Yaskawa INFORM job: X2_55B(90,0).JBI

/JOB
//NAME X2_55B(90,0)
//POS
///NPOS 394,394,394,16,0,0
///TOOL 0
///POSTYPE PULSE
///PULSE
C00000=3322,-122452,-100913,-73,83322,449
C00001=-186633,-49441,-49230,37711,87728,-55120
C00002=-175086,-27134,-34976,36439,84930,-51244
C00003=-172101,-26870,-32446,36082,82517,-50807
C00004=-170908,-26670,-31367,35943,81558,-50627
C00005=-169791,-28532,-32653,35785,80956,-50361
C00006=-170908,-26670,-31367,35943,81558,-50627
C00007=-170104,-28160,-32639,35819,81236,-50399
C00008=-170107,-27903,-30796,35900,80418,-50669
C00009=-170104,-28160,-32639,35819,81236,-50399
C00010=-170752,-27064,-31161,35943,81224,-50672
C00011=-169656,-24122,-29101,35757,80964,-50300
C00012=-170752,-27064,-31161,35943,81224,-50672
C00013=-171397,-28056,-32227,36028,81614,-50812
C00014=-174408,-28429,-34833,36375,84032,-51262
C00015=-173676,-39982,-43344,21171,57836,-56527
C00016=-171324,-36683,-38335,20265,55943,-55912
C00017=-170409,-35305,-36277,19908,55192,-55668
C00018=-170412,-34971,-34390,20145,54260,-55855
C00019=-170409,-35305,-36277,19908,55192,-55668
C00020=-170406,-35026,-34613,20115,54362,-55832
C00021=-168977,-33998,-33935,19313,54123,-55256
C00022=-170406,-35026,-34613,20115,54362,-55832
C00023=-171322,-36428,-36691,20470,55114,-56078
C00024=-173675,-39790,-41746,21371,57009,-56697
C00025=-185662,-62363,-56229,27773,58122,-61625
C00026=-182957,-37243,-22211,38142,77839,-57028
C00027=-174986,-21904,-11817,37450,75534,-54407
C00028=-172006,-20811,-8603,37402,73103,-53977
C00029=-171589,-19133,-6407,37448,72531,-54000
C00030=-170468,-20788,-7609,37359,71957,-53715
C00031=-171113,-19844,-6927,37410,72288,-53878
C00032=-171113,-19561,-6133,37473,72012,-53977
C00033=-171113,-19098,-4854,37577,71571,-54137
C00034=-171113,-19354,-5558,37520,71812,-54050
C00035=-170785,-16593,-3525,37458,71805,-53909
C00036=-169831,-14075,-1633,37337,71498,-53600
C00037=-170747,-16496,-3451,37453,71794,-53895
C00038=-172938,-18790,-5592,37628,72854,-54473
C00039=-174418,-22969,-11095,37549,74492,-54531
C00040=-173590,-36455,-27464,23265,50415,-58157
C00041=-171241,-32608,-21983,22436,48472,-57522
C00042=-170327,-31009,-19725,22109,47697,-57271
C00043=-170330,-30281,-17521,22452,46786,-57499
C00044=-170327,-31009,-19725,22109,47697,-57271
C00045=-170446,-30448,-17835,22480,46917,-57523
C00046=-169016,-29467,-17169,21618,46622,-56894
C00047=-170446,-30448,-17835,22480,46917,-57523
C00048=-171361,-32070,-20116,22801,47697,-57774
C00049=-173714,-35969,-25651,23617,49653,-58408
C00050=-187157,-59404,-40892,31105,51702,-64292
C00051=-182523,-36435,-21722,38111,77739,-56877
C00052=-175053,-21948,-11876,37454,75574,-54422
C00053=-172072,-20861,-8666,37406,73142,-53992
C00054=-170880,-20336,-7310,37391,72173,-53819
C00055=-169763,-22108,-8585,37302,71589,-53539
C00056=-170880,-20336,-7310,37391,72173,-53819
C00057=-163968,-30963,-18249,28546,65432,-52550
C00058=-163972,-30194,-16010,28759,64566,-52785
C00059=-171828,-19900,-6902,37491,72561,-54096
C00060=-170589,-16767,-4601,37336,72180,-53691
C00061=-169762,-14573,-2957,37230,71916,-53424
C00062=-170465,-16446,-4362,37321,72141,-53651
C00063=-172082,-18613,-7207,37365,73353,-53922
C00064=-174410,-22968,-11093,37549,74488,-54529
C00065=-173630,-36453,-27441,23290,50415,-58176
C00066=-171279,-32607,-21961,22462,48470,-57541
C00067=-170365,-31009,-19703,22136,47695,-57290
C00068=-170369,-30280,-17499,22478,46784,-57519
C00069=-170365,-31009,-19703,22136,47695,-57290
C00070=-170401,-30398,-17823,22448,46922,-57500
C00071=-168973,-29415,-17155,21586,46628,-56872
C00072=-170401,-30398,-17823,22448,46922,-57500
C00073=-171316,-32020,-20104,22769,47702,-57751
C00074=-173667,-35921,-25640,23585,49656,-58385
C00075=-184061,-55077,-38542,29439,51265,-62922
C00076=-181525,-34817,-20609,38049,77416,-56562
C00077=-175168,-22294,-12057,37473,75570,-54473
C00078=-172179,-21211,-8851,37428,73136,-54041
C00079=-164934,-20244,-11943,27524,72736,-50675
C00080=-164934,-19832,-10624,27608,72202,-50807
C00081=-164934,-20244,-11943,27524,72736,-50675
C00082=-170788,-19176,-6081,37413,72004,-53840
C00083=-170137,-20123,-6769,37360,71672,-53674
C00084=-170788,-19176,-6081,37413,72004,-53840
C00085=-170451,-17518,-5131,37330,72072,-53666
C00086=-169581,-15212,-3412,37215,71799,-53383
C00087=-170948,-17530,-5209,37372,72321,-53796
C00088=-174379,-22994,-11157,37542,74495,-54513
C00089=-173696,-36532,-27476,23332,50416,-58207
C00090=-171343,-32688,-21999,22504,48471,-57571
C00091=-170428,-31090,-19742,22178,47695,-57320
C00092=-170432,-30361,-17538,22521,46785,-57549
C00093=-170428,-31090,-19742,22178,47695,-57320
C00094=-170423,-30483,-17896,22460,46929,-57509
C00095=-168993,-29501,-17229,21598,46634,-56880
C00096=-170423,-30483,-17896,22460,46929,-57509
C00097=-171339,-32105,-20177,22781,47708,-57760
C00098=-173691,-36004,-25710,23598,49663,-58395
C00099=-183961,-54871,-38414,29383,51253,-62877
C00100=-182126,-35603,-21062,38091,77581,-56762
C00101=-175140,-21971,-11768,37472,75549,-54468
C00102=-172157,-20885,-8559,37428,73117,-54039
C00103=-170965,-20360,-7203,37414,72147,-53865
C00104=-169849,-22134,-8479,37326,71562,-53586
C00105=-170965,-20360,-7203,37414,72147,-53865
C00106=-165310,-29694,-17403,28817,66009,-52954
C00107=-165310,-29050,-15538,28988,65287,-53150
C00108=-171258,-19918,-6523,37477,72118,-54004
C00109=-170426,-17807,-4979,37371,71866,-53731
C00110=-169380,-15031,-2910,37233,71539,-53391
C00111=-169955,-16574,-4065,37309,71721,-53578
C00112=-171522,-16229,-3810,37460,72416,-54014
C00113=-174416,-22925,-11129,37542,74526,-54518
C00114=-173673,-36450,-27429,23316,50421,-58195
C00115=-171322,-32606,-21950,22488,48476,-57560
C00116=-170407,-31008,-19692,22162,47701,-57309
C00117=-170411,-30279,-17488,22505,46790,-57538
C00118=-170407,-31008,-19692,22162,47701,-57309
C00119=-170394,-30411,-17842,22442,46925,-57496
C00120=-168966,-29428,-17174,21580,46631,-56867
C00121=-170394,-30411,-17842,22442,46925,-57496
C00122=-171309,-32033,-20124,22763,47705,-57746
C00123=-173661,-35933,-25659,23580,49659,-58381
C00124=-177896,-47999,-50685,14899,88109,-20692
C00125=-171474,-13387,-32995,26955,87451,38414
C00126=-170968,-26590,-20653,68029,76629,42851
C00127=-168455,-24364,-16087,68284,74284,42470
C00128=-167462,-23391,-14189,68413,73355,42312
C00129=-167464,-22868,-12535,68611,73063,41980
C00130=-167462,-23391,-14189,68413,73355,42312
C00131=-167480,-22950,-12770,68584,73114,42023
C00132=-166431,-22389,-12367,68541,72426,42185
C00133=-167480,-22950,-12770,68584,73114,42023
C00134=-168474,-23944,-14688,68443,74043,42183
C00135=-170987,-26223,-19303,68160,76387,42569
C00136=-178015,-29196,-22452,68319,81266,41791
C00137=-175959,-27390,-21216,68244,79952,42141
C00138=-170916,-26575,-20647,68026,76596,42860
C00139=-168404,-24346,-16079,68281,74252,42479
C00140=-167411,-23372,-14181,68410,73322,42321
C00141=-167413,-22850,-12527,68608,73031,41989
C00142=-167411,-23372,-14181,68410,73322,42321
C00143=-167520,-22976,-12785,68586,73139,42016
C00144=-166471,-22416,-12382,68543,72450,42177
C00145=-167520,-22976,-12785,68586,73139,42016
C00146=-168514,-23970,-14702,68445,74068,42175
C00147=-171028,-26246,-19314,68163,76412,42561
C00148=-175959,-27390,-21216,68244,79952,42141
C00149=-177250,-26440,-20564,68269,80853,42004
C00150=-170954,-26577,-20655,68027,76623,42856
C00151=-168442,-24351,-16088,68281,74278,42475
C00152=-167449,-23792,-15537,68251,73591,42590
C00153=-167449,-23537,-14700,68349,73439,42422
C00154=-167449,-23792,-15537,68251,73591,42590
C00155=-166070,-22339,-14503,68155,72712,42832
C00156=-167449,-23792,-15537,68251,73591,42590
C00157=-168444,-23916,-14658,68443,74021,42185
C00158=-170956,-26197,-19274,68160,76364,42572
C00159=-177250,-26440,-20564,68269,80853,42004
C00160=-175728,-25304,-19738,68213,79861,42242
C00161=-170992,-26689,-20702,68035,76638,42839
C00162=-168478,-24463,-16136,68290,74291,42458
C00163=-167484,-23490,-14239,68419,73362,42300
C00164=-167486,-22966,-12584,68617,73070,41968
C00165=-167484,-23490,-14239,68419,73362,42300
C00166=-167481,-23030,-12848,68582,73118,42026
C00167=-166432,-22469,-12445,68539,72429,42188
C00168=-167481,-23030,-12848,68582,73118,42026
C00169=-168476,-24024,-14766,68441,74047,42186
C00170=-170989,-26302,-19378,68159,76391,42571
C00171=-175728,-25304,-19738,68213,79861,42242
C00172=-176618,-29227,-22045,73488,80077,41536
C00173=-172161,-28800,-21751,73383,76996,42032
C00174=-169385,-26618,-17509,73648,74607,41659
C00175=-167563,-23815,-14727,73682,73258,41735
C00176=-167563,-23156,-12665,73937,72973,41305
C00177=-167563,-23556,-13902,73784,73143,41560
C00178=-166501,-22641,-13252,73745,72429,41707
C00179=-167563,-23556,-13902,73784,73143,41560
C00180=-169398,-26250,-16243,73794,74434,41390
C00181=-172174,-28475,-20524,73502,76822,41766
C00182=-176618,-29227,-22045,73488,80077,41536
C00183=-177511,-5639,371,68424,86651,39750
C00184=-171440,-3456,2150,68562,82586,40567
C00185=-170157,619,6666,68653,81457,40444
C00186=-168331,1234,8338,68777,79954,40379
C00187=-168046,-2076,5678,68790,79736,40390
C00188=-167728,-5916,2555,68804,79503,40409
C00189=-167295,-9898,-598,68829,79172,40420
C00190=-166925,-12748,-2804,68854,78881,40421
C00191=-166573,-15365,-4788,68879,78593,40412
C00192=-169406,-16219,-7074,68798,80759,41235
C00193=-170164,-17729,-8787,68449,80176,51061
C00194=-175136,-9519,-2527,68339,83654,50553
C00195=-174791,2460,6527,68482,84972,40271
C00196=-171445,-3730,1370,68530,82722,40712
C00197=-169192,-1950,5863,68774,80488,40214
C00198=-167748,2520,10895,68924,79213,40058
C00199=-167367,-1794,7418,68947,78922,40075
C00200=-166938,-6982,3161,68992,77768,40277
C00201=-166250,-13921,-2117,69275,75344,44273
C00202=-165956,-15478,-3367,69159,75947,48234
C00203=-167609,-17034,-5893,68702,77907,50786
C00204=-170169,-18009,-9551,68404,80308,51201
C00205=-175223,-9646,-3183,68312,83847,50686
C00206=-174908,3052,7586,68499,84915,40106
C00207=-171434,-3401,2195,68562,82582,40568
C00208=-169182,-1586,6724,68821,80349,40067
C00209=-168625,2129,10992,68937,79702,39832
C00210=-168158,-2892,6969,68968,79346,39846
C00211=-167877,-6432,4056,69014,78297,40037
C00212=-167656,-9030,2010,69063,77269,40197
C00213=-167278,-12997,-1111,69137,75067,40567
C00214=-166927,-16034,-3407,69190,73221,40852
C00215=-166736,-17163,-4204,69214,73333,40784
C00216=-166964,-12102,-1327,68082,78867,40243
C00217=-166860,-10009,379,67974,81306,39758
C00218=-167599,-16670,-5060,68761,77774,50646
C00219=-170158,-17675,-8747,68448,80173,51063
C00220=-175928,-7987,-1318,68319,84203,50466
C00221=-174129,1419,6201,68516,84397,40216
C00222=-171443,-3483,2127,68562,82588,40566
C00223=-169190,-1670,6655,68820,80354,40066
C00224=-168618,1929,10819,68939,79695,39833
C00225=-168181,-3083,6692,68956,79389,39875
C00226=-167825,-6908,3653,69018,78263,40044
C00227=-167628,-9346,1685,69056,77267,40218
C00228=-167197,-13163,-1220,69143,75004,40568
C00229=-166871,-15927,-3321,69191,73184,40859
C00230=-166710,-17179,-4282,69204,73330,40804
C00231=-166618,-17311,-4405,69161,75321,40414
C00232=-167253,-2768,6900,68495,85595,38662
C00233=-167607,-16752,-5121,68762,77778,50643
C00234=-170167,-17757,-8807,68449,80178,51060
C00235=-175992,-7969,-1304,68317,84246,50458
C00236=-174493,2196,6858,68508,84639,40165
C00237=-171437,-3428,2172,68562,82584,40568
C00238=-169184,-1614,6701,68820,80351,40067
C00239=-168608,2565,11412,68945,79676,39815
C00240=-168131,-2876,6882,68959,79351,39876
C00241=-167879,-6487,3954,69009,78311,40050
C00242=-167834,-6567,3889,69012,78225,40066
C00243=-167304,-13008,-1155,69131,75092,40573
C00244=-167217,-13136,-1253,69134,74889,40610
C00245=-166739,-17203,-4252,69210,73342,40789
C00246=-166985,-13978,-1962,69009,77711,40070
C00247=-167253,-4374,5575,68532,84778,38834
C00248=-168446,-14711,-4185,68664,78524,50736
C00249=-170161,-17702,-8767,68449,80174,51062
C00250=-175232,-9311,-2363,68337,83721,50543
C00251=-175249,13254,-9292,16869,97733,1178
C00252=-168597,-48257,-56117,1181,80760,-43912
C00253=-177620,-43084,-26025,45113,44922,-82367
C00254=-174971,-39401,-20697,44915,42590,-82091
C00255=-174605,-35611,-17109,44939,42219,-82082
C00256=-174724,-34541,-16405,44907,42364,-82069
C00257=-177051,-29782,-13235,47611,46397,-84220
C00258=-177434,-27688,-11867,47614,46759,-84238
C00259=-177667,-25419,-10216,47598,46981,-84242
C00260=-178185,-29641,-14356,47538,47518,-84232
C00261=-180753,-32756,-19483,47484,49943,-84329
C00262=-173287,-17819,-8789,22973,65327,-48793
C00263=-170946,-14881,-3560,22677,63099,-48320
C00264=-169599,-10626,768,22411,62289,-47944
C00265=-167576,-15676,-2878,20525,60168,-45587
C00266=-167052,-17460,-4261,20372,59975,-45406
C00267=-166529,-18969,-5372,20230,59762,-45234
C00268=-167807,-11208,-706,22629,68741,-42434
C00269=-169790,-14055,-4135,22891,69883,-42970
C00270=-172168,-16723,-9131,23082,72120,-43433
C00271=-171866,-14901,-7113,34634,81390,-68840
C00272=-169482,-15346,-4516,34706,78904,-68641
C00273=-167855,-13991,-2244,34715,77661,-68363
C00274=-167135,-12229,-875,34671,77417,-68142
C00275=-166013,-9105,1504,34599,77077,-67783
C00276=-166134,-13157,-36,37044,72073,-67632
C00277=-167931,-14988,-2581,37092,73349,-67963
C00278=-170473,-15229,-5631,37029,75857,-68181
C00279=-178233,-32689,-17977,37632,78114,-70716
C00280=-188699,-64462,-48311,47699,52584,-74036
C00281=-177600,-47289,-38890,41459,49172,-79942
C00282=-174952,-43987,-33928,40953,46886,-79574
C00283=-174398,-40381,-30434,40853,46398,-79496
C00284=-174619,-39339,-29742,40991,46666,-79594
C00285=-175378,-38206,-29028,42112,47956,-80386
C00286=-176767,-35152,-27115,43849,50364,-81644
C00287=-177145,-32637,-25411,43890,50728,-81667
C00288=-177529,-29433,-23171,43905,51114,-81681
C00289=-178167,-33843,-27515,43948,51733,-81719
C00290=-180735,-36508,-32225,44206,54131,-81906
C00291=-173238,-22685,-36674,21290,78953,-46169
C00292=-170900,-20986,-32518,20780,76785,-45705
C00293=-170144,-18859,-29851,20614,76082,-45550
C00294=-168456,-23469,-33122,18801,74180,-43497
C00295=-167647,-26136,-35012,18575,73801,-43261
C00296=-166864,-28508,-36654,18360,73428,-43034
C00297=-168669,-18522,-30713,21504,82655,-40150
C00298=-168439,-19208,-31172,21461,82531,-40087
C00299=-169745,-19576,-32646,21691,83540,-40375
C00300=-172121,-21002,-36582,22105,85735,-40825
C00301=-171835,-19421,-31884,34437,92133,-65504
C00302=-169453,-21055,-30238,34176,89639,-65313
C00303=-168630,-22241,-29853,34096,88606,-65296
C00304=-167284,-18647,-27256,33962,88272,-64858
C00305=-166994,-18189,-26846,34071,87788,-64721
C00306=-166806,-21636,-27949,35609,82808,-64307
C00307=-167902,-21345,-28846,35726,83840,-64426
C00308=-170444,-20454,-30963,36019,86338,-64655
C00309=-177146,-36799,-42202,36823,87959,-66885
C00310=-189885,-60568,-35825,51532,49461,-81920
C00311=-177609,-43032,-25994,45103,44922,-82360
C00312=-174962,-39349,-20664,44906,42590,-82085
C00313=-174429,-35406,-16945,44857,42132,-82023
C00314=-176890,-30423,-13789,47560,46319,-84168
C00315=-177369,-28075,-12315,47519,46779,-84182
C00316=-177701,-25498,-10475,47531,47083,-84200
C00317=-178175,-29589,-14321,47530,47517,-84226
C00318=-180742,-32704,-19449,47476,49941,-84323
C00319=-173279,-17766,-8750,22970,65328,-48790
C00320=-170939,-14827,-3519,22675,63100,-48317
C00321=-169374,-10615,423,22306,62431,-47826
C00322=-168875,-12851,-1454,22165,62303,-47648
C00323=-168243,-14554,-2565,22032,61954,-47466
C00324=-167157,-18210,-5323,21764,61497,-47117
C00325=-167721,-10961,-888,22579,68936,-42365
C00326=-169783,-14001,-4094,22890,69884,-42968
C00327=-172161,-16669,-9091,23080,72121,-43430
C00328=-171868,-14843,-7099,34633,81408,-68835
C00329=-169486,-15291,-4504,34704,78924,-68637
C00330=-167771,-14162,-2743,34687,77809,-68281
C00331=-167071,-12040,-1190,34635,77630,-68045
C00332=-165773,-8384,1630,34554,77222,-67639
C00333=-166155,-12879,-165,37009,72266,-67573
C00334=-167935,-14934,-2570,37088,73368,-67958
C00335=-170477,-15173,-5619,37026,75875,-68176
C00336=-177184,-30600,-16616,37567,77846,-70362
C00337=-190085,-60834,-35962,51621,49539,-82793
C00338=-177625,-43110,-26041,45118,44922,-82371
C00339=-174976,-39427,-20713,44920,42590,-82094
C00340=-174545,-35598,-17276,44832,42266,-82011
C00341=-174667,-35018,-16914,44830,42381,-82019
C00342=-177022,-29976,-13569,47545,46457,-84165
C00343=-177431,-27692,-12033,47527,46829,-84187
C00344=-177751,-25532,-10543,47514,47131,-84199
C00345=-178190,-29666,-14374,47541,47519,-84234
C00346=-180759,-32781,-19500,47487,49944,-84332
C00347=-173290,-17849,-8819,22973,65331,-48794
C00348=-170949,-14912,-3590,22677,63103,-48320
C00349=-170097,-9297,1554,22507,62609,-48083
C00350=-169747,-10570,589,22423,62460,-47969
C00351=-169007,-13054,-1319,22242,62165,-47729
C00352=-168006,-16287,-3803,21993,61775,-47405
C00353=-168148,-11038,-697,22541,67989,-43198
C00354=-169793,-14086,-4166,22891,69887,-42971
C00355=-172172,-16753,-9161,23082,72124,-43434
C00356=-171879,-14924,-7160,34633,81409,-68839
C00357=-169495,-15372,-4565,34705,78924,-68641
C00358=-168548,-12947,-1667,34723,78094,-68514
C00359=-167717,-10836,16,34683,77796,-68263
C00360=-166486,-7202,2727,34603,77460,-67860
C00361=-170164,-14497,2537,44164,69716,-72995
C00362=-167944,-15015,-2632,37090,73368,-67961
C00363=-170486,-15254,-5680,37027,75876,-68179
C00364=-177884,-32016,-17561,37610,78034,-70595
C00365=-191188,-62009,-36562,52066,50005,-77650
C00366=-177614,-43058,-26010,45108,44922,-82364
C00367=-174966,-39375,-20681,44911,42590,-82088
C00368=-174503,-35547,-17229,44808,42247,-81997
C00369=-174586,-34848,-16787,44787,42346,-81987
C00370=-176974,-29345,-13125,47472,46466,-84124
C00371=-177351,-26855,-11354,47501,46793,-84158
C00372=-177581,-25325,-10300,47504,47011,-84167
C00373=-178180,-29615,-14339,47534,47518,-84229
C00374=-180748,-32730,-19466,47480,49942,-84326
C00375=-173283,-17792,-8769,22971,65327,-48791
C00376=-170942,-14854,-3539,22676,63100,-48318
C00377=-170055,-9124,1558,22476,62681,-48045
C00378=-169100,-12658,-1111,22253,62260,-47746
C00379=-168593,-14307,-2366,22128,62054,-47584
C00380=-167713,-16948,-4365,21909,61702,-47298
C00381=-172853,-2835,7813,29766,72471,-47128
C00382=-169787,-14028,-4114,22890,69884,-42969
C00383=-172165,-16696,-9111,23081,72121,-43432
C00384=-171872,-14870,-7119,34633,81408,-68836
C00385=-169489,-15318,-4525,34704,78924,-68638
C00386=-168322,-12820,-1688,34704,78074,-68432
C00387=-167882,-11409,-693,34676,77989,-68276
C00388=-166167,-6498,3088,34573,77457,-67736
C00389=-170486,-15775,2354,45649,68509,-73783
C00390=-167938,-14961,-2591,37089,73368,-67959
C00391=-170480,-15200,-5639,37027,75875,-68177
C00392=-178859,-33825,-18753,37663,78302,-70918
C00393=3322,-122452,-100913,-73,83322,449
BC00000=87761,666220,1075229
BC00001=92219,666220,1075175
BC00002=92219,666220,1075175
BC00003=92219,666220,1075175
BC00004=92219,666220,1075175
BC00005=92219,666220,1075175
BC00006=92219,666220,1075175
BC00007=92219,666220,1075175
BC00008=92219,666220,1075175
BC00009=92219,666220,1075175
BC00010=92219,666220,1075175
BC00011=92219,666220,1075175
BC00012=92219,666220,1075175
BC00013=92219,666220,1075175
BC00014=92219,666220,1075175
BC00015=117428,666220,1075175
BC00016=117428,666220,1075175
BC00017=117428,666220,1075175
BC00018=117428,666220,1075175
BC00019=117428,666220,1075175
BC00020=117428,666220,1075175
BC00021=117428,666220,1075175
BC00022=117428,666220,1075175
BC00023=117428,666220,1075175
BC00024=117428,666220,1075175
BC00025=117428,666220,1075175
BC00026=92232,666220,1039532
BC00027=92232,666220,1039532
BC00028=92232,666220,1039532
BC00029=92232,666220,1039532
BC00030=92232,666220,1039532
BC00031=92232,666220,1039532
BC00032=92232,666220,1039532
BC00033=92232,666220,1039532
BC00034=92232,666220,1039532
BC00035=92232,666220,1039532
BC00036=92232,666220,1039532
BC00037=92232,666220,1039532
BC00038=92232,666220,1039532
BC00039=92232,666220,1039532
BC00040=117405,666220,1001297
BC00041=117405,666220,1001297
BC00042=117405,666220,1001297
BC00043=117405,666220,1001297
BC00044=117405,666220,1001297
BC00045=117405,666220,1001297
BC00046=117405,666220,1001297
BC00047=117405,666220,1001297
BC00048=117405,666220,1001297
BC00049=117405,666220,1001297
BC00050=117405,666220,1001297
BC00051=92302,666220,877583
BC00052=92302,666220,877583
BC00053=92302,666220,877583
BC00054=92302,666220,877583
BC00055=92302,666220,877583
BC00056=92302,666220,877583
BC00057=92302,666220,877583
BC00058=92302,666220,877583
BC00059=92302,666220,877583
BC00060=92302,666220,877583
BC00061=92302,666220,877583
BC00062=92302,666220,877583
BC00063=92302,666220,877583
BC00064=92302,666220,877583
BC00065=117238,666220,839321
BC00066=117238,666220,839321
BC00067=117238,666220,839321
BC00068=117238,666220,839321
BC00069=117238,666220,839321
BC00070=117238,666220,839321
BC00071=117238,666220,839321
BC00072=117238,666220,839321
BC00073=117238,666220,839321
BC00074=117238,666220,839321
BC00075=117238,666220,839321
BC00076=92181,666220,715340
BC00077=92181,666220,715340
BC00078=92181,666220,715340
BC00079=92181,666220,715340
BC00080=92181,666220,715340
BC00081=92181,666220,715340
BC00082=92181,666220,715340
BC00083=92181,666220,715340
BC00084=92181,666220,715340
BC00085=92181,666220,715340
BC00086=92181,666220,715340
BC00087=92181,666220,715340
BC00088=92181,666220,715340
BC00089=117409,666220,677313
BC00090=117409,666220,677313
BC00091=117409,666220,677313
BC00092=117409,666220,677313
BC00093=117409,666220,677313
BC00094=117409,666220,677313
BC00095=117409,666220,677313
BC00096=117409,666220,677313
BC00097=117409,666220,677313
BC00098=117409,666220,677313
BC00099=117409,666220,677313
BC00100=92362,666220,553818
BC00101=92362,666220,553818
BC00102=92362,666220,553818
BC00103=92362,666220,553818
BC00104=92362,666220,553818
BC00105=92362,666220,553818
BC00106=92362,666220,553818
BC00107=92362,666220,553818
BC00108=92362,666220,553818
BC00109=92362,666220,553818
BC00110=92362,666220,553818
BC00111=92362,666220,553818
BC00112=92362,666220,553818
BC00113=92362,666220,553818
BC00114=117290,666220,515979
BC00115=117290,666220,515979
BC00116=117290,666220,515979
BC00117=117290,666220,515979
BC00118=117290,666220,515979
BC00119=117290,666220,515979
BC00120=117290,666220,515979
BC00121=117290,666220,515979
BC00122=117290,666220,515979
BC00123=117290,666220,515979
BC00124=87994,666220,479725
BC00125=36377,666220,415849
BC00126=28007,666220,405491
BC00127=28007,666220,405491
BC00128=28007,666220,405491
BC00129=28007,666220,405491
BC00130=28007,666220,405491
BC00131=28007,666220,405491
BC00132=28007,666220,405491
BC00133=28007,666220,405491
BC00134=28007,666220,405491
BC00135=28007,666220,405491
BC00136=28007,666220,405491
BC00137=28126,666220,566762
BC00138=28126,666220,566762
BC00139=28126,666220,566762
BC00140=28126,666220,566762
BC00141=28126,666220,566762
BC00142=28126,666220,566762
BC00143=28126,666220,566762
BC00144=28126,666220,566762
BC00145=28126,666220,566762
BC00146=28126,666220,566762
BC00147=28126,666220,566762
BC00148=28126,666220,566762
BC00149=27845,666220,728834
BC00150=27845,666220,728834
BC00151=27845,666220,728834
BC00152=27845,666220,728834
BC00153=27845,666220,728834
BC00154=27845,666220,728834
BC00155=27845,666220,728834
BC00156=27845,666220,728834
BC00157=27845,666220,728834
BC00158=27845,666220,728834
BC00159=27845,666220,728834
BC00160=27967,666220,891139
BC00161=27967,666220,891139
BC00162=27967,666220,891139
BC00163=27967,666220,891139
BC00164=27967,666220,891139
BC00165=27967,666220,891139
BC00166=27967,666220,891139
BC00167=27967,666220,891139
BC00168=27967,666220,891139
BC00169=27967,666220,891139
BC00170=27967,666220,891139
BC00171=27967,666220,891139
BC00172=25231,666220,1022271
BC00173=25231,666220,1022271
BC00174=25231,666220,1022271
BC00175=25231,666220,1022270
BC00176=25231,666220,1022271
BC00177=25231,666220,1022271
BC00178=25231,666220,1022271
BC00179=25231,666220,1022271
BC00180=25231,666220,1022271
BC00181=25231,666220,1022271
BC00182=25231,666220,1022271
BC00183=27733,666220,754462
BC00184=27733,666220,754462
BC00185=27733,666220,754462
BC00186=27733,666220,754462
BC00187=27733,666220,754462
BC00188=27733,666220,754462
BC00189=27733,666220,754462
BC00190=27733,666220,754462
BC00191=27733,666220,754462
BC00192=27733,666220,754462
BC00193=27733,666220,754462
BC00194=27733,666220,754462
BC00195=27726,666220,1075175
BC00196=27726,666220,1075175
BC00197=27726,666220,1075175
BC00198=27726,666220,1075175
BC00199=27726,666220,1075175
BC00200=27726,666220,1075175
BC00201=27726,666220,1075175
BC00202=27726,666220,1075175
BC00203=27726,666220,1075175
BC00204=27726,666220,1075175
BC00205=27726,666220,1075175
BC00206=27740,666220,431052
BC00207=27740,666220,431052
BC00208=27740,666220,431052
BC00209=27740,666220,431052
BC00210=27740,666220,431052
BC00211=27740,666220,431052
BC00212=27740,666220,431052
BC00213=27740,666220,431052
BC00214=27740,666220,431052
BC00215=27740,666220,431052
BC00216=27740,666220,431052
BC00217=27740,666220,431052
BC00218=27740,666220,431052
BC00219=27740,666220,431052
BC00220=27740,666220,431052
BC00221=27730,666220,916571
BC00222=27730,666220,916571
BC00223=27730,666220,916571
BC00224=27730,666220,916571
BC00225=27730,666220,916571
BC00226=27730,666220,916571
BC00227=27730,666220,916571
BC00228=27730,666220,916571
BC00229=27730,666220,916571
BC00230=27730,666220,916571
BC00231=27730,666220,916571
BC00232=27730,666220,916571
BC00233=27730,666220,916571
BC00234=27730,666220,916571
BC00235=27730,666220,916571
BC00236=27736,666220,592354
BC00237=27736,666220,592354
BC00238=27736,666220,592354
BC00239=27736,666220,592354
BC00240=27736,666220,592354
BC00241=27736,666220,592354
BC00242=27736,666220,592354
BC00243=27736,666220,592354
BC00244=27736,666220,592354
BC00245=27736,666220,592354
BC00246=27736,666221,592352
BC00247=27736,666221,592352
BC00248=27736,666220,592354
BC00249=27736,666220,592354
BC00250=27736,666220,592354
BC00251=66745,666220,695171
BC00252=94472,666220,768252
BC00253=112638,666220,816133
BC00254=112638,666220,816133
BC00255=112638,666220,816133
BC00256=112638,666220,816133
BC00257=112638,666220,816133
BC00258=112638,666220,816133
BC00259=112638,666220,816133
BC00260=112638,666220,816133
BC00261=112638,666220,816133
BC00262=117812,666220,907206
BC00263=117812,666220,907206
BC00264=117812,666220,907206
BC00265=117812,666220,907206
BC00266=117812,666220,907206
BC00267=117812,666220,907206
BC00268=117812,666220,907206
BC00269=117812,666220,907206
BC00270=117812,666220,907206
BC00271=87729,666220,888327
BC00272=87729,666220,888327
BC00273=87729,666220,888327
BC00274=87729,666220,888327
BC00275=87729,666220,888327
BC00276=87729,666220,888327
BC00277=87729,666220,888327
BC00278=87729,666220,888327
BC00279=87729,666220,888327
BC00280=112631,666220,1075175
BC00281=112631,666220,1075175
BC00282=112631,666220,1075175
BC00283=112631,666220,1075175
BC00284=112631,666220,1075175
BC00285=112631,666220,1075175
BC00286=112631,666220,1075175
BC00287=112631,666220,1075175
BC00288=112631,666220,1075175
BC00289=112631,666220,1075175
BC00290=112631,666220,1075175
BC00291=117805,666220,1075175
BC00292=117805,666220,1075175
BC00293=117805,666220,1075175
BC00294=117805,666220,1075175
BC00295=117805,666220,1075175
BC00296=117805,666220,1075175
BC00297=117805,666220,1075175
BC00298=117805,666220,1075175
BC00299=117805,666220,1075175
BC00300=117805,666220,1075175
BC00301=87751,666220,1075175
BC00302=87751,666220,1075175
BC00303=87751,666221,1075173
BC00304=87751,666220,1075175
BC00305=87751,666220,1075175
BC00306=87751,666220,1075175
BC00307=87751,666220,1075175
BC00308=87751,666220,1075175
BC00309=87751,666220,1075175
BC00310=112645,666220,492722
BC00311=112645,666220,492722
BC00312=112645,666220,492722
BC00313=112645,666220,492722
BC00314=112645,666220,492722
BC00315=112645,666220,492722
BC00316=112645,666220,492722
BC00317=112645,666220,492722
BC00318=112645,666220,492722
BC00319=117819,666220,583796
BC00320=117819,666220,583796
BC00321=117819,666220,583796
BC00322=117819,666220,583796
BC00323=117819,666220,583796
BC00324=117819,666220,583796
BC00325=117819,666220,583796
BC00326=117819,666220,583796
BC00327=117819,666220,583796
BC00328=87764,666220,564729
BC00329=87764,666220,564729
BC00330=87764,666220,564729
BC00331=87764,666220,564729
BC00332=87764,666220,564729
BC00333=87764,666220,564729
BC00334=87764,666220,564729
BC00335=87764,666220,564729
BC00336=87764,666220,564729
BC00337=112635,666220,978242
BC00338=112635,666220,978242
BC00339=112635,666220,978242
BC00340=112635,666220,978242
BC00341=112635,666220,978242
BC00342=112635,666220,978242
BC00343=112635,666220,978242
BC00344=112635,666220,978242
BC00345=112635,666220,978242
BC00346=112635,666220,978242
BC00347=117809,666220,1069266
BC00348=117809,666220,1069266
BC00349=117809,666220,1069266
BC00350=117809,666220,1069266
BC00351=117809,666220,1069266
BC00352=117809,666220,1069266
BC00353=117808,666220,1069263
BC00354=117809,666220,1069266
BC00355=117809,666220,1069266
BC00356=87754,666220,1050249
BC00357=87754,666220,1050249
BC00358=87754,666220,1050249
BC00359=87754,666220,1050249
BC00360=87754,666220,1050249
BC00361=87754,666220,1050249
BC00362=87754,666220,1050249
BC00363=87754,666220,1050249
BC00364=87754,666220,1050249
BC00365=112641,666220,654024
BC00366=112641,666220,654024
BC00367=112641,666220,654024
BC00368=112641,666220,654024
BC00369=112641,666220,654024
BC00370=112641,666220,654024
BC00371=112641,666220,654024
BC00372=112641,666220,654024
BC00373=112641,666220,654024
BC00374=112641,666220,654024
BC00375=117815,666220,745098
BC00376=117815,666220,745098
BC00377=117815,666220,745098
BC00378=117815,666220,745098
BC00379=117815,666220,745098
BC00380=117815,666220,745098
BC00381=117815,666220,745098
BC00382=117815,666220,745098
BC00383=117815,666220,745098
BC00384=87761,666220,726031
BC00385=87761,666220,726031
BC00386=87761,666220,726031
BC00387=87761,666220,726031
BC00388=87761,666220,726031
BC00389=87761,666220,726031
BC00390=87761,666220,726031
BC00391=87761,666220,726031
BC00392=87761,666220,726031
BC00393=87761,666220,1075229
EC00000=798156,0
EC00001=798156,0
EC00002=798156,0
EC00003=798156,0
EC00004=798156,0
EC00005=798156,0
EC00006=798156,0
EC00007=798156,0
EC00008=798156,0
EC00009=798156,0
EC00010=798156,0
EC00011=798156,0
EC00012=798156,0
EC00013=798156,0
EC00014=798156,0
EC00015=798156,0
EC00016=798156,0
EC00017=798156,0
EC00018=798156,0
EC00019=798156,0
EC00020=798156,0
EC00021=798156,0
EC00022=798156,0
EC00023=798156,0
EC00024=798156,0
EC00025=798156,0
EC00026=798156,0
EC00027=798156,0
EC00028=798156,0
EC00029=798156,0
EC00030=798156,0
EC00031=798156,0
EC00032=798156,0
EC00033=798156,0
EC00034=798156,0
EC00035=798156,0
EC00036=798156,0
EC00037=798156,0
EC00038=798156,0
EC00039=798156,0
EC00040=798156,0
EC00041=798156,0
EC00042=798156,0
EC00043=798156,0
EC00044=798156,0
EC00045=798156,0
EC00046=798156,0
EC00047=798156,0
EC00048=798156,0
EC00049=798156,0
EC00050=798156,0
EC00051=798156,0
EC00052=798156,0
EC00053=798156,0
EC00054=798156,0
EC00055=798156,0
EC00056=798156,0
EC00057=798156,0
EC00058=798156,0
EC00059=798156,0
EC00060=798156,0
EC00061=798156,0
EC00062=798156,0
EC00063=798156,0
EC00064=798156,0
EC00065=798156,0
EC00066=798156,0
EC00067=798156,0
EC00068=798156,0
EC00069=798156,0
EC00070=798156,0
EC00071=798156,0
EC00072=798156,0
EC00073=798156,0
EC00074=798156,0
EC00075=798156,0
EC00076=798156,0
EC00077=798156,0
EC00078=798156,0
EC00079=798156,0
EC00080=798156,0
EC00081=798156,0
EC00082=798156,0
EC00083=798156,0
EC00084=798156,0
EC00085=798156,0
EC00086=798156,0
EC00087=798156,0
EC00088=798156,0
EC00089=798156,0
EC00090=798156,0
EC00091=798156,0
EC00092=798156,0
EC00093=798156,0
EC00094=798156,0
EC00095=798156,0
EC00096=798156,0
EC00097=798156,0
EC00098=798156,0
EC00099=798156,0
EC00100=798156,0
EC00101=798156,0
EC00102=798156,0
EC00103=798156,0
EC00104=798156,0
EC00105=798156,0
EC00106=798156,0
EC00107=798156,0
EC00108=798156,0
EC00109=798156,0
EC00110=798156,0
EC00111=798156,0
EC00112=798156,0
EC00113=798156,0
EC00114=798156,0
EC00115=798156,0
EC00116=798156,0
EC00117=798156,0
EC00118=798156,0
EC00119=798156,0
EC00120=798156,0
EC00121=798156,0
EC00122=798156,0
EC00123=798156,0
EC00124=798156,0
EC00125=798156,0
EC00126=798156,0
EC00127=798156,0
EC00128=798156,0
EC00129=798156,0
EC00130=798156,0
EC00131=798156,0
EC00132=798156,0
EC00133=798156,0
EC00134=798156,0
EC00135=798156,0
EC00136=798156,0
EC00137=798156,0
EC00138=798156,0
EC00139=798156,0
EC00140=798156,0
EC00141=798156,0
EC00142=798156,0
EC00143=798156,0
EC00144=798156,0
EC00145=798156,0
EC00146=798156,0
EC00147=798156,0
EC00148=798156,0
EC00149=798156,0
EC00150=798156,0
EC00151=798156,0
EC00152=798156,0
EC00153=798156,0
EC00154=798156,0
EC00155=798156,0
EC00156=798156,0
EC00157=798156,0
EC00158=798156,0
EC00159=798156,0
EC00160=798156,0
EC00161=798156,0
EC00162=798156,0
EC00163=798156,0
EC00164=798156,0
EC00165=798156,0
EC00166=798156,0
EC00167=798156,0
EC00168=798156,0
EC00169=798156,0
EC00170=798156,0
EC00171=798156,0
EC00172=798156,0
EC00173=798156,0
EC00174=798156,0
EC00175=798153,1
EC00176=798156,0
EC00177=798156,0
EC00178=798156,0
EC00179=798156,0
EC00180=798156,0
EC00181=798156,0
EC00182=798156,0
EC00183=798156,0
EC00184=798156,0
EC00185=798156,0
EC00186=798156,0
EC00187=798156,0
EC00188=798156,0
EC00189=798156,0
EC00190=798156,0
EC00191=798156,0
EC00192=798156,0
EC00193=798156,0
EC00194=798156,0
EC00195=798156,0
EC00196=798156,0
EC00197=798156,0
EC00198=798156,0
EC00199=798156,0
EC00200=798156,0
EC00201=798156,0
EC00202=798156,0
EC00203=798156,0
EC00204=798156,0
EC00205=798156,0
EC00206=798156,0
EC00207=798156,0
EC00208=798156,0
EC00209=798156,0
EC00210=798156,0
EC00211=798156,0
EC00212=798156,0
EC00213=798156,0
EC00214=798156,0
EC00215=798156,0
EC00216=798156,0
EC00217=798156,0
EC00218=798156,0
EC00219=798156,0
EC00220=798156,0
EC00221=798156,0
EC00222=798156,0
EC00223=798156,0
EC00224=798156,0
EC00225=798156,0
EC00226=798156,0
EC00227=798156,0
EC00228=798156,0
EC00229=798156,0
EC00230=798156,0
EC00231=798156,0
EC00232=798156,0
EC00233=798156,0
EC00234=798156,0
EC00235=798156,0
EC00236=798156,0
EC00237=798156,0
EC00238=798156,0
EC00239=798156,0
EC00240=798156,0
EC00241=798156,0
EC00242=798156,0
EC00243=798156,0
EC00244=798156,0
EC00245=798156,0
EC00246=798155,0
EC00247=798155,0
EC00248=798156,0
EC00249=798156,0
EC00250=798156,0
EC00251=798156,0
EC00252=798156,0
EC00253=798156,0
EC00254=798156,0
EC00255=798156,0
EC00256=798156,0
EC00257=798156,0
EC00258=798156,0
EC00259=798156,0
EC00260=798156,0
EC00261=798156,0
EC00262=798156,0
EC00263=798156,0
EC00264=798156,0
EC00265=798156,0
EC00266=798156,0
EC00267=798156,0
EC00268=798156,0
EC00269=798156,0
EC00270=798156,0
EC00271=798156,0
EC00272=798156,0
EC00273=798156,0
EC00274=798156,0
EC00275=798156,0
EC00276=798156,0
EC00277=798156,0
EC00278=798156,0
EC00279=798156,0
EC00280=798156,0
EC00281=798156,0
EC00282=798156,0
EC00283=798156,0
EC00284=798156,0
EC00285=798156,0
EC00286=798156,0
EC00287=798156,0
EC00288=798156,0
EC00289=798156,0
EC00290=798156,0
EC00291=798156,0
EC00292=798156,0
EC00293=798156,0
EC00294=798156,0
EC00295=798156,0
EC00296=798156,0
EC00297=798156,0
EC00298=798156,0
EC00299=798156,0
EC00300=798156,0
EC00301=798156,0
EC00302=798156,0
EC00303=798155,1
EC00304=798156,0
EC00305=798156,0
EC00306=798156,0
EC00307=798156,0
EC00308=798156,0
EC00309=798156,0
EC00310=798156,0
EC00311=798156,0
EC00312=798156,0
EC00313=798156,0
EC00314=798156,0
EC00315=798156,0
EC00316=798156,0
EC00317=798156,0
EC00318=798156,0
EC00319=798156,0
EC00320=798156,0
EC00321=798156,0
EC00322=798156,0
EC00323=798156,0
EC00324=798156,0
EC00325=798156,0
EC00326=798156,0
EC00327=798156,0
EC00328=798156,0
EC00329=798156,0
EC00330=798156,0
EC00331=798156,0
EC00332=798156,0
EC00333=798156,0
EC00334=798156,0
EC00335=798156,0
EC00336=798156,0
EC00337=798156,0
EC00338=798156,0
EC00339=798156,0
EC00340=798156,0
EC00341=798156,0
EC00342=798156,0
EC00343=798156,0
EC00344=798156,0
EC00345=798156,0
EC00346=798156,0
EC00347=798156,0
EC00348=798156,0
EC00349=798156,0
EC00350=798156,0
EC00351=798156,0
EC00352=798156,0
EC00353=798154,1
EC00354=798156,0
EC00355=798156,0
EC00356=798156,0
EC00357=798156,0
EC00358=798156,0
EC00359=798156,0
EC00360=798156,0
EC00361=798156,0
EC00362=798156,0
EC00363=798156,0
EC00364=798156,0
EC00365=798156,0
EC00366=798156,0
EC00367=798156,0
EC00368=798156,0
EC00369=798156,0
EC00370=798156,0
EC00371=798156,0
EC00372=798156,0
EC00373=798156,0
EC00374=798156,0
EC00375=798156,0
EC00376=798156,0
EC00377=798156,0
EC00378=798156,0
EC00379=798156,0
EC00380=798156,0
EC00381=798156,0
EC00382=798156,0
EC00383=798156,0
EC00384=798156,0
EC00385=798156,0
EC00386=798156,0
EC00387=798156,0
EC00388=798156,0
EC00389=798156,0
EC00390=798156,0
EC00391=798156,0
EC00392=798156,0
EC00393=798156,0
///POSTYPE BASE
///RECTAN
///RCONF 0,0,0,0,0,0,0,0,0,0,0,0,0,0,0,0,0,0,0,0,0,0,0,0
P00006=0.222,-3.123,-1.508,0.0000,0.0000,0.0000
P00021=-0.225,-6.128,-0.405,0.0000,0.0000,0.0000
P00022=0.222,-3.123,-1.508,0.0000,0.0000,0.0000
P00023=0.143,-0.036,0.682,0.0000,0.0000,0.0000
P00031=1.853,-0.001,-1.549,0.0000,0.0000,0.0000
P00032=1.957,0.503,-7.217,0.0000,0.0000,0.0000
///RCONF 0,0,0,0,1,0,0,0,0,0,0,0,0,0,0,0,0,0,0,0,0,0,0,0
P00033=-0.123,0.612,-5.012,0.0000,0.0000,0.0000
///RCONF 0,0,0,0,0,0,0,0,0,0,0,0,0,0,0,0,0,0,0,0,0,0,0,0
P00041=0.192,3.924,0.305,0.0000,0.0000,0.0000
P00042=-0.217,1.941,0.413,0.0000,0.0000,0.0000
P00043=-0.044,-1.937,1.197,0.0000,0.0000,0.0000
P00051=0.367,3.892,0.009,0.0000,0.0000,0.0000
P00052=0.088,2.832,-0.342,0.0000,0.0000,0.0000
P00053=0.134,6.594,0.107,0.0000,0.0000,0.0000
P00061=1.575,-3.405,-0.752,0.0000,0.0000,0.0000
P00062=-0.135,-0.848,-1.706,0.0000,0.0000,0.0000
P00063=0.036,-0.654,-3.005,0.0000,0.0000,0.0000
//INST
///DATE 2024/11/18 13:39
///ATTR SC,RW
///GROUP1 RB1,BS1
///GROUP2 ST1
NOP
'X2_55b(90,0)
'
MOVJ C00000 BC00000 VJ=100.00  +MOVJ EC00000 VJ=100.00
MOVJ C00001 BC00001 VJ=100.00  +MOVJ EC00001 VJ=100.00
'Path S4425
SFTOF3D
MOVJ C00002 BC00002 VJ=100.00  +MOVJ EC00002 VJ=100.00
MOVL C00003 BC00003 V=800.0  +MOVJ EC00003 VJ=100.00
SMOVL C00004 BC00004 V=166.7  +MOVJ EC00004
SREFP 3 C00005 BC00005  +REFP EC00005
CALL JOB:SEARCH-R1-S13D
SET P021 P006
SFTON3D P021
SMOVL C00006 BC00006 V=166.7  +MOVJ EC00006
SMOVL C00007 BC00007 V=166.7  +MOVJ EC00007
SREFP 3 C00008 BC00008  +REFP EC00008
CALL JOB:SEARCH-R1-S13D
SET P021 P006
SFTON3D P021
SMOVL C00009 BC00009 V=166.7  +MOVJ EC00009
SMOVL C00010 BC00010 V=166.7  +MOVJ EC00010
SREFP 3 C00011 BC00011  +REFP EC00011
CALL JOB:SEARCH-R1-S13D
SET P021 P006
SFTON3D P021
SMOVL C00012 BC00012 V=166.7  +MOVJ EC00012
MOVL C00013 BC00013 V=800.0  +MOVJ EC00013 VJ=100.00
MOVL C00014 BC00014 V=1000.0  +MOVJ EC00014 VJ=100.00
'EndPath S4425
'Path S4426
SFTOF3D
MOVJ C00015 BC00015 VJ=100.00  +MOVJ EC00015 VJ=100.00
MOVL C00016 BC00016 V=800.0  +MOVJ EC00016 VJ=100.00
SMOVL C00017 BC00017 V=166.7  +MOVJ EC00017
SREFP 3 C00018 BC00018  +REFP EC00018
CALL JOB:SEARCH-R1-S13D
SET P022 P006
SFTON3D P022
SMOVL C00019 BC00019 V=166.7  +MOVJ EC00019
SMOVL C00020 BC00020 V=166.7  +MOVJ EC00020
SREFP 3 C00021 BC00021  +REFP EC00021
CALL JOB:SEARCH-R1-S13D
SET P022 P006
SFTON3D P022
SMOVL C00022 BC00022 V=166.7  +MOVJ EC00022
MOVL C00023 BC00023 V=800.0  +MOVJ EC00023 VJ=100.00
MOVL C00024 BC00024 V=1000.0  +MOVJ EC00024 VJ=100.00
'EndPath S4426
MOVJ C00025 BC00025 VJ=100.00  +MOVJ EC00025 VJ=100.00
'
MOVJ C00026 BC00026 VJ=100.00  +MOVJ EC00026 VJ=100.00
'Path S4427
SFTOF3D
MOVJ C00027 BC00027 VJ=100.00  +MOVJ EC00027 VJ=100.00
MOVL C00028 BC00028 V=800.0  +MOVJ EC00028 VJ=100.00
SMOVL C00029 BC00029 V=166.7  +MOVJ EC00029
SREFP 3 C00030 BC00030  +REFP EC00030
CALL JOB:SEARCH-R1-S13D
SET P031 P006
SFTON3D P031
SMOVL C00031 BC00031 V=166.7  +MOVJ EC00031
SMOVL C00032 BC00032 V=166.7  +MOVJ EC00032
SREFP 3 C00033 BC00033  +REFP EC00033
CALL JOB:SEARCH-R1-S13D
SET P031 P006
SFTON3D P031
SMOVL C00034 BC00034 V=166.7  +MOVJ EC00034
SMOVL C00035 BC00035 V=166.7  +MOVJ EC00035
SREFP 3 C00036 BC00036  +REFP EC00036
CALL JOB:SEARCH-R1-S13D
SET P031 P006
SFTON3D P031
SMOVL C00037 BC00037 V=166.7  +MOVJ EC00037
MOVL C00038 BC00038 V=800.0  +MOVJ EC00038 VJ=100.00
MOVL C00039 BC00039 V=1000.0  +MOVJ EC00039 VJ=100.00
'EndPath S4427
'Path S4428
SFTOF3D
MOVJ C00040 BC00040 VJ=100.00  +MOVJ EC00040 VJ=100.00
MOVL C00041 BC00041 V=800.0  +MOVJ EC00041 VJ=100.00
SMOVL C00042 BC00042 V=166.7  +MOVJ EC00042
SREFP 3 C00043 BC00043  +REFP EC00043
CALL JOB:SEARCH-R1-S13D
SET P032 P006
SFTON3D P032
SMOVL C00044 BC00044 V=166.7  +MOVJ EC00044
SMOVL C00045 BC00045 V=166.7  +MOVJ EC00045
SREFP 3 C00046 BC00046  +REFP EC00046
CALL JOB:SEARCH-R1-S13D
SET P032 P006
SFTON3D P032
SMOVL C00047 BC00047 V=166.7  +MOVJ EC00047
MOVL C00048 BC00048 V=800.0  +MOVJ EC00048 VJ=100.00
MOVL C00049 BC00049 V=1000.0  +MOVJ EC00049 VJ=100.00
'EndPath S4428
MOVJ C00050 BC00050 VJ=100.00  +MOVJ EC00050 VJ=100.00
'
MOVJ C00051 BC00051 VJ=100.00  +MOVJ EC00051 VJ=100.00
'Path S4429
SFTOF3D
MOVJ C00052 BC00052 VJ=100.00  +MOVJ EC00052 VJ=100.00
MOVL C00053 BC00053 V=800.0  +MOVJ EC00053 VJ=100.00
SMOVL C00054 BC00054 V=166.7  +MOVJ EC00054
SREFP 3 C00055 BC00055  +REFP EC00055
CALL JOB:SEARCH-R1-S13D
SET P041 P006
SFTON3D P041
SMOVL C00056 BC00056 V=166.7  +MOVJ EC00056
SMOVL C00057 BC00057 V=166.7  +MOVJ EC00057
SREFP 3 C00058 BC00058  +REFP EC00058
CALL JOB:SEARCH-R1-S13D
SET P041 P006
SFTON3D P041
SMOVL C00059 BC00059 V=166.7  +MOVJ EC00059
SMOVL C00060 BC00060 V=166.7  +MOVJ EC00060
SREFP 3 C00061 BC00061  +REFP EC00061
CALL JOB:SEARCH-R1-S13D
SET P041 P006
SFTON3D P041
SMOVL C00062 BC00062 V=166.7  +MOVJ EC00062
MOVL C00063 BC00063 V=800.0  +MOVJ EC00063 VJ=100.00
MOVL C00064 BC00064 V=1000.0  +MOVJ EC00064 VJ=100.00
'EndPath S4429
'Path S4430
SFTOF3D
MOVJ C00065 BC00065 VJ=100.00  +MOVJ EC00065 VJ=100.00
MOVL C00066 BC00066 V=800.0  +MOVJ EC00066 VJ=100.00
SMOVL C00067 BC00067 V=166.7  +MOVJ EC00067
SREFP 3 C00068 BC00068  +REFP EC00068
CALL JOB:SEARCH-R1-S13D
SET P042 P006
SFTON3D P042
SMOVL C00069 BC00069 V=166.7  +MOVJ EC00069
SMOVL C00070 BC00070 V=166.7  +MOVJ EC00070
SREFP 3 C00071 BC00071  +REFP EC00071
CALL JOB:SEARCH-R1-S13D
SET P042 P006
SFTON3D P042
SMOVL C00072 BC00072 V=166.7  +MOVJ EC00072
MOVL C00073 BC00073 V=800.0  +MOVJ EC00073 VJ=100.00
MOVL C00074 BC00074 V=1000.0  +MOVJ EC00074 VJ=100.00
'EndPath S4430
MOVJ C00075 BC00075 VJ=100.00  +MOVJ EC00075 VJ=100.00
'
MOVJ C00076 BC00076 VJ=100.00  +MOVJ EC00076 VJ=100.00
'Path S4431
SFTOF3D
MOVJ C00077 BC00077 VJ=100.00  +MOVJ EC00077 VJ=100.00
MOVL C00078 BC00078 V=800.0  +MOVJ EC00078 VJ=100.00
SMOVL C00079 BC00079 V=166.7  +MOVJ EC00079
SREFP 3 C00080 BC00080  +REFP EC00080
CALL JOB:SEARCH-R1-S13D
SET P051 P006
SFTON3D P051
SMOVL C00081 BC00081 V=166.7  +MOVJ EC00081
SMOVL C00082 BC00082 V=166.7  +MOVJ EC00082
SREFP 3 C00083 BC00083  +REFP EC00083
CALL JOB:SEARCH-R1-S13D
SET P051 P006
SFTON3D P051
SMOVL C00084 BC00084 V=166.7  +MOVJ EC00084
SMOVL C00085 BC00085 V=166.7  +MOVJ EC00085
SREFP 3 C00086 BC00086  +REFP EC00086
CALL JOB:SEARCH-R1-S13D
SET P051 P006
SFTON3D P051
SMOVL C00087 BC00087 V=250.0  +MOVJ EC00087
MOVL C00088 BC00088 V=1000.0  +MOVJ EC00088 VJ=100.00
'EndPath S4431
'Path S4432
SFTOF3D
MOVJ C00089 BC00089 VJ=100.00  +MOVJ EC00089 VJ=100.00
MOVL C00090 BC00090 V=800.0  +MOVJ EC00090 VJ=100.00
SMOVL C00091 BC00091 V=166.7  +MOVJ EC00091
SREFP 3 C00092 BC00092  +REFP EC00092
CALL JOB:SEARCH-R1-S13D
SET P052 P006
SFTON3D P052
SMOVL C00093 BC00093 V=166.7  +MOVJ EC00093
SMOVL C00094 BC00094 V=166.7  +MOVJ EC00094
SREFP 3 C00095 BC00095  +REFP EC00095
CALL JOB:SEARCH-R1-S13D
SET P052 P006
SFTON3D P052
SMOVL C00096 BC00096 V=166.7  +MOVJ EC00096
MOVL C00097 BC00097 V=800.0  +MOVJ EC00097 VJ=100.00
MOVL C00098 BC00098 V=1000.0  +MOVJ EC00098 VJ=100.00
'EndPath S4432
MOVJ C00099 BC00099 VJ=100.00  +MOVJ EC00099 VJ=100.00
'
MOVJ C00100 BC00100 VJ=100.00  +MOVJ EC00100 VJ=100.00
'Path S4433
SFTOF3D
MOVJ C00101 BC00101 VJ=100.00  +MOVJ EC00101 VJ=100.00
MOVL C00102 BC00102 V=800.0  +MOVJ EC00102 VJ=100.00
SMOVL C00103 BC00103 V=166.7  +MOVJ EC00103
SREFP 3 C00104 BC00104  +REFP EC00104
CALL JOB:SEARCH-R1-S13D
SET P061 P006
SFTON3D P061
SMOVL C00105 BC00105 V=166.7  +MOVJ EC00105
SMOVL C00106 BC00106 V=166.7  +MOVJ EC00106
SREFP 3 C00107 BC00107  +REFP EC00107
CALL JOB:SEARCH-R1-S13D
SET P061 P006
SFTON3D P061
SMOVL C00108 BC00108 V=166.7  +MOVJ EC00108
SMOVL C00109 BC00109 V=166.7  +MOVJ EC00109
SREFP 3 C00110 BC00110  +REFP EC00110
CALL JOB:SEARCH-R1-S13D
SET P061 P006
SFTON3D P061
SMOVL C00111 BC00111 V=166.7  +MOVJ EC00111
MOVL C00112 BC00112 V=800.0  +MOVJ EC00112 VJ=100.00
MOVL C00113 BC00113 V=1000.0  +MOVJ EC00113 VJ=100.00
'EndPath S4433
'Path S4434
SFTOF3D
MOVJ C00114 BC00114 VJ=100.00  +MOVJ EC00114 VJ=100.00
MOVL C00115 BC00115 V=800.0  +MOVJ EC00115 VJ=100.00
SMOVL C00116 BC00116 V=166.7  +MOVJ EC00116
SREFP 3 C00117 BC00117  +REFP EC00117
CALL JOB:SEARCH-R1-S13D
SET P062 P006
SFTON3D P062
SMOVL C00118 BC00118 V=166.7  +MOVJ EC00118
SMOVL C00119 BC00119 V=166.7  +MOVJ EC00119
SREFP 3 C00120 BC00120  +REFP EC00120
CALL JOB:SEARCH-R1-S13D
SET P062 P006
SFTON3D P062
SMOVL C00121 BC00121 V=166.7  +MOVJ EC00121
MOVL C00122 BC00122 V=800.0  +MOVJ EC00122 VJ=100.00
MOVL C00123 BC00123 V=1000.0  +MOVJ EC00123 VJ=100.00
'EndPath S4434
MOVJ C00124 BC00124 VJ=100.00  +MOVJ EC00124 VJ=100.00
MOVJ C00125 BC00125 VJ=100.00  +MOVJ EC00125 VJ=100.00
'
'Path S4435
SFTOF3D
MOVJ C00126 BC00126 VJ=100.00  +MOVJ EC00126 VJ=100.00
MOVL C00127 BC00127 V=800.0  +MOVJ EC00127 VJ=100.00
SMOVL C00128 BC00128 V=166.7  +MOVJ EC00128
SREFP 3 C00129 BC00129  +REFP EC00129
CALL JOB:SEARCH-R1-S13D
SET P063 P006
SFTON3D P063
SMOVL C00130 BC00130 V=166.7  +MOVJ EC00130
SMOVL C00131 BC00131 V=166.7  +MOVJ EC00131
SREFP 3 C00132 BC00132  +REFP EC00132
CALL JOB:SEARCH-R1-S13D
SET P063 P006
SFTON3D P063
SMOVL C00133 BC00133 V=166.7  +MOVJ EC00133
MOVL C00134 BC00134 V=800.0  +MOVJ EC00134 VJ=100.00
MOVL C00135 BC00135 V=1000.0  +MOVJ EC00135 VJ=100.00
'EndPath S4435
MOVJ C00136 BC00136 VJ=100.00  +MOVJ EC00136 VJ=100.00
MOVJ C00137 BC00137 VJ=100.00  +MOVJ EC00137 VJ=100.00
'Path S4436
SFTOF3D
MOVJ C00138 BC00138 VJ=100.00  +MOVJ EC00138 VJ=100.00
MOVL C00139 BC00139 V=800.0  +MOVJ EC00139 VJ=100.00
SMOVL C00140 BC00140 V=166.7  +MOVJ EC00140
SREFP 3 C00141 BC00141  +REFP EC00141
CALL JOB:SEARCH-R1-S13D
SET P053 P006
SFTON3D P053
SMOVL C00142 BC00142 V=166.7  +MOVJ EC00142
SMOVL C00143 BC00143 V=166.7  +MOVJ EC00143
SREFP 3 C00144 BC00144  +REFP EC00144
CALL JOB:SEARCH-R1-S13D
SET P053 P006
SFTON3D P053
SMOVL C00145 BC00145 V=166.7  +MOVJ EC00145
MOVL C00146 BC00146 V=800.0  +MOVJ EC00146 VJ=100.00
MOVL C00147 BC00147 V=1000.0  +MOVJ EC00147 VJ=100.00
'EndPath S4436
MOVJ C00148 BC00148 VJ=100.00  +MOVJ EC00148 VJ=100.00
MOVJ C00149 BC00149 VJ=100.00  +MOVJ EC00149 VJ=100.00
'Path S4437
SFTOF3D
MOVJ C00150 BC00150 VJ=100.00  +MOVJ EC00150 VJ=100.00
MOVL C00151 BC00151 V=800.0  +MOVJ EC00151 VJ=100.00
SMOVL C00152 BC00152 V=166.7  +MOVJ EC00152
SREFP 3 C00153 BC00153  +REFP EC00153
CALL JOB:SEARCH-R1-S13D
SET P043 P006
SFTON3D P043
SMOVL C00154 BC00154 V=166.7  +MOVJ EC00154
SREFP 3 C00155 BC00155  +REFP EC00155
CALL JOB:SEARCH-R1-S13D
SET P043 P006
SFTON3D P043
SMOVL C00156 BC00156 V=166.7  +MOVJ EC00156
MOVL C00157 BC00157 V=800.0  +MOVJ EC00157 VJ=100.00
MOVL C00158 BC00158 V=1000.0  +MOVJ EC00158 VJ=100.00
'EndPath S4437
MOVJ C00159 BC00159 VJ=100.00  +MOVJ EC00159 VJ=100.00
MOVJ C00160 BC00160 VJ=100.00  +MOVJ EC00160 VJ=100.00
'Path S4438
SFTOF3D
MOVJ C00161 BC00161 VJ=100.00  +MOVJ EC00161 VJ=100.00
MOVL C00162 BC00162 V=800.0  +MOVJ EC00162 VJ=100.00
SMOVL C00163 BC00163 V=166.7  +MOVJ EC00163
SREFP 3 C00164 BC00164  +REFP EC00164
CALL JOB:SEARCH-R1-S13D
SET P033 P006
SFTON3D P033
SMOVL C00165 BC00165 V=166.7  +MOVJ EC00165
SMOVL C00166 BC00166 V=166.7  +MOVJ EC00166
SREFP 3 C00167 BC00167  +REFP EC00167
CALL JOB:SEARCH-R1-S13D
SET P033 P006
SFTON3D P033
SMOVL C00168 BC00168 V=166.7  +MOVJ EC00168
MOVL C00169 BC00169 V=800.0  +MOVJ EC00169 VJ=100.00
MOVL C00170 BC00170 V=1000.0  +MOVJ EC00170 VJ=100.00
'EndPath S4438
MOVJ C00171 BC00171 VJ=100.00  +MOVJ EC00171 VJ=100.00
MOVJ C00172 BC00172 VJ=100.00  +MOVJ EC00172 VJ=100.00
'Path S4439
SFTOF3D
MOVJ C00173 BC00173 VJ=100.00  +MOVJ EC00173 VJ=100.00
MOVL C00174 BC00174 V=800.0  +MOVJ EC00174 VJ=100.00
SMOVL C00175 BC00175 V=166.7  +MOVJ EC00175
SREFP 3 C00176 BC00176  +REFP EC00176
CALL JOB:SEARCH-R1-S13D
SET P023 P006
SFTON3D P023
SMOVL C00177 BC00177 V=166.7  +MOVJ EC00177
SREFP 3 C00178 BC00178  +REFP EC00178
CALL JOB:SEARCH-R1-S13D
SET P023 P006
SFTON3D P023
SMOVL C00179 BC00179 V=166.7  +MOVJ EC00179
MOVL C00180 BC00180 V=800.0  +MOVJ EC00180 VJ=100.00
MOVL C00181 BC00181 V=1000.0  +MOVJ EC00181 VJ=100.00
'EndPath S4439
MOVJ C00182 BC00182 VJ=100.00  +MOVJ EC00182 VJ=100.00
'
'
'
MOVJ C00183 BC00183 VJ=100.00  +MOVJ EC00183 VJ=100.00
'Path W4440
SFTOF3D
SFTON3D P043
MOVJ C00184 BC00184 VJ=100.00  +MOVJ EC00184 VJ=100.00
SMOVL C00185 BC00185 V=800.0  +MOVJ EC00185
SMOVL C00186 BC00186 V=166.7 PL=0  +MOVJ EC00186
ARCON
SMOVL C00187 BC00187 V=10.0  +MOVJ EC00187
SMOVL C00188 BC00188 V=10.0  +MOVJ EC00188
SMOVL C00189 BC00189 V=10.0  +MOVJ EC00189
SMOVL C00190 BC00190 V=10.0  +MOVJ EC00190
SMOVL C00191 BC00191 V=10.0  +MOVJ EC00191
ARCOF
SMOVL C00192 BC00192 V=800.0  +MOVJ EC00192
SMOVL C00193 BC00193 V=1000.0  +MOVJ EC00193
SFTOF3D
'EndPath W4440
MOVJ C00194 BC00194 VJ=100.00  +MOVJ EC00194 VJ=100.00
MOVJ C00195 BC00195 VJ=100.00  +MOVJ EC00195 VJ=100.00
'Path W4441
SFTOF3D
SFTON3D P023
MOVJ C00196 BC00196 VJ=100.00  +MOVJ EC00196 VJ=100.00
SMOVL C00197 BC00197 V=800.0  +MOVJ EC00197
SMOVL C00198 BC00198 V=166.7 PL=0  +MOVJ EC00198
ARCON
SMOVL C00199 BC00199 V=10.0  +MOVJ EC00199
SMOVL C00200 BC00200 V=10.0  +MOVJ EC00200
SMOVL C00201 BC00201 V=10.0  +MOVJ EC00201
SMOVL C00202 BC00202 V=10.0  +MOVJ EC00202
ARCOF
SMOVL C00203 BC00203 V=800.0  +MOVJ EC00203
SMOVL C00204 BC00204 V=1000.0  +MOVJ EC00204
SFTOF3D
'EndPath W4441
MOVJ C00205 BC00205 VJ=100.00  +MOVJ EC00205 VJ=100.00
MOVJ C00206 BC00206 VJ=100.00  +MOVJ EC00206 VJ=100.00
'Path W4442
SFTOF3D
SFTON3D P063
MOVJ C00207 BC00207 VJ=100.00  +MOVJ EC00207 VJ=100.00
SMOVL C00208 BC00208 V=800.0  +MOVJ EC00208
SMOVL C00209 BC00209 V=166.7 PL=0  +MOVJ EC00209
ARCON
SMOVL C00210 BC00210 V=10.0  +MOVJ EC00210
SMOVL C00211 BC00211 V=10.0  +MOVJ EC00211
SMOVL C00212 BC00212 V=10.0  +MOVJ EC00212
SMOVL C00213 BC00213 V=10.0  +MOVJ EC00213
SMOVL C00214 BC00214 V=10.0  +MOVJ EC00214
SMOVL C00215 BC00215 V=10.0  +MOVJ EC00215
SMOVL C00216 BC00216 V=10.0  +MOVJ EC00216
SMOVL C00217 BC00217 V=10.0  +MOVJ EC00217
ARCOF
SMOVL C00218 BC00218 V=800.0  +MOVJ EC00218
SMOVL C00219 BC00219 V=1000.0  +MOVJ EC00219
SFTOF3D
'EndPath W4442
MOVJ C00220 BC00220 VJ=100.00  +MOVJ EC00220 VJ=100.00
MOVJ C00221 BC00221 VJ=100.00  +MOVJ EC00221 VJ=100.00
'Path W4443
SFTOF3D
SFTON3D P033
MOVJ C00222 BC00222 VJ=100.00  +MOVJ EC00222 VJ=100.00
SMOVL C00223 BC00223 V=800.0  +MOVJ EC00223
SMOVL C00224 BC00224 V=166.7 PL=0  +MOVJ EC00224
ARCON
SMOVL C00225 BC00225 V=10.0  +MOVJ EC00225
SMOVL C00226 BC00226 V=10.0  +MOVJ EC00226
SMOVL C00227 BC00227 V=10.0  +MOVJ EC00227
SMOVL C00228 BC00228 V=10.0  +MOVJ EC00228
SMOVL C00229 BC00229 V=10.0  +MOVJ EC00229
SMOVL C00230 BC00230 V=10.0  +MOVJ EC00230
SMOVL C00231 BC00231 V=10.0  +MOVJ EC00231
SMOVL C00232 BC00232 V=10.0  +MOVJ EC00232
ARCOF
SMOVL C00233 BC00233 V=800.0  +MOVJ EC00233
SMOVL C00234 BC00234 V=1000.0  +MOVJ EC00234
SFTOF3D
'EndPath W4443
MOVJ C00235 BC00235 VJ=100.00  +MOVJ EC00235 VJ=100.00
MOVJ C00236 BC00236 VJ=100.00  +MOVJ EC00236 VJ=100.00
'Path W4444
SFTOF3D
SFTON3D P053
MOVJ C00237 BC00237 VJ=100.00  +MOVJ EC00237 VJ=100.00
SMOVL C00238 BC00238 V=800.0  +MOVJ EC00238
SMOVL C00239 BC00239 V=166.7 PL=0  +MOVJ EC00239
ARCON
SMOVL C00240 BC00240 V=10.0  +MOVJ EC00240
SMOVL C00241 BC00241 V=10.0  +MOVJ EC00241
SMOVL C00242 BC00242 V=10.0  +MOVJ EC00242
SMOVL C00243 BC00243 V=10.0  +MOVJ EC00243
SMOVL C00244 BC00244 V=10.0  +MOVJ EC00244
SMOVL C00245 BC00245 V=10.0  +MOVJ EC00245
SMOVL C00246 BC00246 V=10.0  +MOVJ EC00246
SMOVL C00247 BC00247 V=10.0  +MOVJ EC00247
ARCOF
SMOVL C00248 BC00248 V=800.0  +MOVJ EC00248
SMOVL C00249 BC00249 V=1000.0  +MOVJ EC00249
SFTOF3D
'EndPath W4444
MOVJ C00250 BC00250 VJ=100.00  +MOVJ EC00250 VJ=100.00
'
MOVJ C00251 BC00251 VJ=100.00  +MOVJ EC00251 VJ=100.00
MOVJ C00252 BC00252 VJ=100.00  +MOVJ EC00252 VJ=100.00
'Path W4445
SFTOF3D
SFTON3D P042
MOVJ C00253 BC00253 VJ=100.00  +MOVJ EC00253 VJ=100.00
SMOVL C00254 BC00254 V=800.0  +MOVJ EC00254
SMOVL C00255 BC00255 V=166.7 PL=0  +MOVJ EC00255
ARCON
SMOVL C00256 BC00256 V=10.0  +MOVJ EC00256
SMOVL C00257 BC00257 V=10.0  +MOVJ EC00257
SMOVL C00258 BC00258 V=10.0  +MOVJ EC00258
SMOVL C00259 BC00259 V=10.0  +MOVJ EC00259
ARCOF
SMOVL C00260 BC00260 V=800.0  +MOVJ EC00260
SMOVL C00261 BC00261 V=1000.0  +MOVJ EC00261
SFTOF3D
'EndPath W4445
'Path W4446
SFTOF3D
SFTON3D P041
MOVJ C00262 BC00262 VJ=100.00  +MOVJ EC00262 VJ=100.00
SMOVL C00263 BC00263 V=800.0  +MOVJ EC00263
SMOVL C00264 BC00264 V=166.7 PL=0  +MOVJ EC00264
ARCON
SMOVL C00265 BC00265 V=10.0  +MOVJ EC00265
SMOVL C00266 BC00266 V=10.0  +MOVJ EC00266
SMOVL C00267 BC00267 V=10.0  +MOVJ EC00267
SMOVL C00268 BC00268 V=10.0  +MOVJ EC00268
ARCOF
SMOVL C00269 BC00269 V=800.0  +MOVJ EC00269
SMOVL C00270 BC00270 V=1000.0  +MOVJ EC00270
SFTOF3D
'EndPath W4446
'Path W4447
SFTOF3D
SFTON3D P041
MOVJ C00271 BC00271 VJ=100.00  +MOVJ EC00271 VJ=100.00
SMOVL C00272 BC00272 V=800.0  +MOVJ EC00272
SMOVL C00273 BC00273 V=166.7 PL=0  +MOVJ EC00273
ARCON
SMOVL C00274 BC00274 V=10.0  +MOVJ EC00274
SMOVL C00275 BC00275 V=10.0  +MOVJ EC00275
SMOVL C00276 BC00276 V=10.0  +MOVJ EC00276
ARCOF
SMOVL C00277 BC00277 V=800.0  +MOVJ EC00277
SMOVL C00278 BC00278 V=1000.0  +MOVJ EC00278
SFTOF3D
'EndPath W4447
MOVJ C00279 BC00279 VJ=100.00  +MOVJ EC00279 VJ=100.00
'
'
MOVJ C00280 BC00280 VJ=100.00  +MOVJ EC00280 VJ=100.00
'Path W4448
SFTOF3D
SFTON3D P022
MOVJ C00281 BC00281 VJ=100.00  +MOVJ EC00281 VJ=100.00
SMOVL C00282 BC00282 V=800.0  +MOVJ EC00282
SMOVL C00283 BC00283 V=166.7 PL=0  +MOVJ EC00283
MACRO1 MJ#(0) ARGF9
ARCON
SMOVL C00284 BC00284 V=10.0  +MOVJ EC00284
SMOVL C00285 BC00285 V=10.0  +MOVJ EC00285
SMOVL C00286 BC00286 V=10.0  +MOVJ EC00286
SMOVL C00287 BC00287 V=10.0  +MOVJ EC00287
SMOVL C00288 BC00288 V=10.0  +MOVJ EC00288
ARCOF
SMOVL C00289 BC00289 V=800.0  +MOVJ EC00289
SMOVL C00290 BC00290 V=1000.0  +MOVJ EC00290
SFTOF3D
'EndPath W4448
'Path W4449
SFTOF3D
SFTON3D P021
MOVJ C00291 BC00291 VJ=100.00  +MOVJ EC00291 VJ=100.00
SMOVL C00292 BC00292 V=800.0  +MOVJ EC00292
SMOVL C00293 BC00293 V=166.7 PL=0  +MOVJ EC00293
ARCON
SMOVL C00294 BC00294 V=10.0  +MOVJ EC00294
SMOVL C00295 BC00295 V=10.0  +MOVJ EC00295
SMOVL C00296 BC00296 V=10.0  +MOVJ EC00296
SMOVL C00297 BC00297 V=10.0  +MOVJ EC00297
SMOVL C00298 BC00298 V=10.0  +MOVJ EC00298
ARCOF
SMOVL C00299 BC00299 V=800.0  +MOVJ EC00299
SMOVL C00300 BC00300 V=1000.0  +MOVJ EC00300
SFTOF3D
'EndPath W4449
'Path W4450
SFTOF3D
SFTON3D P021
MOVJ C00301 BC00301 VJ=100.00  +MOVJ EC00301 VJ=100.00
SMOVL C00302 BC00302 V=800.0  +MOVJ EC00302
SMOVL C00303 BC00303 V=166.7 PL=0  +MOVJ EC00303
ARCON
SMOVL C00304 BC00304 V=10.0  +MOVJ EC00304
SMOVL C00305 BC00305 V=10.0  +MOVJ EC00305
SMOVL C00306 BC00306 V=10.0  +MOVJ EC00306
ARCOF
SMOVL C00307 BC00307 V=800.0  +MOVJ EC00307
SMOVL C00308 BC00308 V=1000.0  +MOVJ EC00308
SFTOF3D
'EndPath W4450
MOVJ C00309 BC00309 VJ=100.00  +MOVJ EC00309 VJ=100.00
'
'
MOVJ C00310 BC00310 VJ=100.00  +MOVJ EC00310 VJ=100.00
'Path W4451
SFTOF3D
SFTON3D P062
MOVJ C00311 BC00311 VJ=100.00  +MOVJ EC00311 VJ=100.00
SMOVL C00312 BC00312 V=800.0  +MOVJ EC00312
SMOVL C00313 BC00313 V=166.7 PL=0  +MOVJ EC00313
ARCON
SMOVL C00314 BC00314 V=10.0  +MOVJ EC00314
SMOVL C00315 BC00315 V=10.0  +MOVJ EC00315
SMOVL C00316 BC00316 V=10.0  +MOVJ EC00316
ARCOF
SMOVL C00317 BC00317 V=800.0  +MOVJ EC00317
SMOVL C00318 BC00318 V=1000.0  +MOVJ EC00318
SFTOF3D
'EndPath W4451
'Path W4452
SFTOF3D
SFTON3D P061
MOVJ C00319 BC00319 VJ=100.00  +MOVJ EC00319 VJ=100.00
MACRO1 MJ#(0) ARGF21
SMOVL C00320 BC00320 V=800.0  +MOVJ EC00320
SMOVL C00321 BC00321 V=166.7 PL=0  +MOVJ EC00321
ARCON
SMOVL C00322 BC00322 V=10.0  +MOVJ EC00322
SMOVL C00323 BC00323 V=10.0  +MOVJ EC00323
SMOVL C00324 BC00324 V=10.0  +MOVJ EC00324
SMOVL C00325 BC00325 V=10.0  +MOVJ EC00325
ARCOF
SMOVL C00326 BC00326 V=800.0  +MOVJ EC00326
SMOVL C00327 BC00327 V=1000.0  +MOVJ EC00327
SFTOF3D
'EndPath W4452
'Path W4453
SFTOF3D
SFTON3D P061
MOVJ C00328 BC00328 VJ=100.00  +MOVJ EC00328 VJ=100.00
SMOVL C00329 BC00329 V=800.0  +MOVJ EC00329
SMOVL C00330 BC00330 V=166.7 PL=0  +MOVJ EC00330
ARCON
SMOVL C00331 BC00331 V=10.0  +MOVJ EC00331
SMOVL C00332 BC00332 V=10.0  +MOVJ EC00332
ARCON
SMOVL C00333 BC00333 V=10.0  +MOVJ EC00333
ARCOF
SMOVL C00334 BC00334 V=800.0  +MOVJ EC00334
SMOVL C00335 BC00335 V=1000.0  +MOVJ EC00335
SFTOF3D
'EndPath W4453
MOVJ C00336 BC00336 VJ=100.00  +MOVJ EC00336 VJ=100.00
'
'
MOVJ C00337 BC00337 VJ=100.00  +MOVJ EC00337 VJ=100.00
'Path W4454
SFTOF3D
SFTON3D P032
MOVJ C00338 BC00338 VJ=100.00  +MOVJ EC00338 VJ=100.00
SMOVL C00339 BC00339 V=800.0  +MOVJ EC00339
SMOVL C00340 BC00340 V=166.7 PL=0  +MOVJ EC00340
ARCON
SMOVL C00341 BC00341 V=10.0  +MOVJ EC00341
SMOVL C00342 BC00342 V=10.0  +MOVJ EC00342
SMOVL C00343 BC00343 V=10.0  +MOVJ EC00343
SMOVL C00344 BC00344 V=10.0  +MOVJ EC00344
ARCOF
SMOVL C00345 BC00345 V=800.0  +MOVJ EC00345
SMOVL C00346 BC00346 V=1000.0  +MOVJ EC00346
SFTOF3D
'EndPath W4454
'Path W4455
SFTOF3D
SFTON3D P031
MOVJ C00347 BC00347 VJ=100.00  +MOVJ EC00347 VJ=100.00
SMOVL C00348 BC00348 V=800.0  +MOVJ EC00348
SMOVL C00349 BC00349 V=166.7 PL=0  +MOVJ EC00349
ARCON
SMOVL C00350 BC00350 V=10.0  +MOVJ EC00350
SMOVL C00351 BC00351 V=10.0  +MOVJ EC00351
SMOVL C00352 BC00352 V=10.0  +MOVJ EC00352
SMOVL C00353 BC00353 V=10.0  +MOVJ EC00353
ARCOF
SMOVL C00354 BC00354 V=800.0  +MOVJ EC00354
SMOVL C00355 BC00355 V=1000.0  +MOVJ EC00355
SFTOF3D
'EndPath W4455
'Path W4456
SFTOF3D
SFTON3D P031
MOVJ C00356 BC00356 VJ=100.00  +MOVJ EC00356 VJ=100.00
SMOVL C00357 BC00357 V=800.0  +MOVJ EC00357
SMOVL C00358 BC00358 V=166.7 PL=0  +MOVJ EC00358
ARCON
SMOVL C00359 BC00359 V=10.0  +MOVJ EC00359
SMOVL C00360 BC00360 V=10.0  +MOVJ EC00360
SMOVL C00361 BC00361 V=10.0  +MOVJ EC00361
ARCOF
SMOVL C00362 BC00362 V=800.0  +MOVJ EC00362
SMOVL C00363 BC00363 V=1000.0  +MOVJ EC00363
SFTOF3D
'EndPath W4456
MOVJ C00364 BC00364 VJ=100.00  +MOVJ EC00364 VJ=100.00
'
'
MOVJ C00365 BC00365 VJ=100.00  +MOVJ EC00365 VJ=100.00
'Path W4457
SFTOF3D
SFTON3D P052
MOVJ C00366 BC00366 VJ=100.00  +MOVJ EC00366 VJ=100.00
SMOVL C00367 BC00367 V=800.0  +MOVJ EC00367
MACRO1 MJ#(0) ARGF14
SMOVL C00368 BC00368 V=166.7 PL=0  +MOVJ EC00368
ARCON
SMOVL C00369 BC00369 V=10.0  +MOVJ EC00369
SMOVL C00370 BC00370 V=10.0  +MOVJ EC00370
SMOVL C00371 BC00371 V=10.0  +MOVJ EC00371
SMOVL C00372 BC00372 V=10.0  +MOVJ EC00372
ARCOF
SMOVL C00373 BC00373 V=800.0  +MOVJ EC00373
SMOVL C00374 BC00374 V=1000.0  +MOVJ EC00374
SFTOF3D
'EndPath W4457
'Path W4458
SFTOF3D
SFTON3D P051
MOVJ C00375 BC00375 VJ=100.00  +MOVJ EC00375 VJ=100.00
SMOVL C00376 BC00376 V=800.0  +MOVJ EC00376
MACRO1 MJ#(0) ARGF21
SMOVL C00377 BC00377 V=166.7 PL=0  +MOVJ EC00377
ARCON
SMOVL C00378 BC00378 V=10.0  +MOVJ EC00378
SMOVL C00379 BC00379 V=10.0  +MOVJ EC00379
SMOVL C00380 BC00380 V=10.0  +MOVJ EC00380
SMOVL C00381 BC00381 V=10.0  +MOVJ EC00381
ARCOF
SMOVL C00382 BC00382 V=800.0  +MOVJ EC00382
SMOVL C00383 BC00383 V=1000.0  +MOVJ EC00383
SFTOF3D
'EndPath W4458
'Path W4459
SFTOF3D
SFTON3D P051
MOVJ C00384 BC00384 VJ=100.00  +MOVJ EC00384 VJ=100.00
SMOVL C00385 BC00385 V=800.0  +MOVJ EC00385
SMOVL C00386 BC00386 V=166.7 PL=0  +MOVJ EC00386
ARCON
SMOVL C00387 BC00387 V=10.0  +MOVJ EC00387
SMOVL C00388 BC00388 V=10.0  +MOVJ EC00388
SMOVL C00389 BC00389 V=10.0  +MOVJ EC00389
ARCOF
SMOVL C00390 BC00390 V=800.0  +MOVJ EC00390
SMOVL C00391 BC00391 V=1000.0  +MOVJ EC00391
SFTOF3D
'EndPath W4459
MOVJ C00392 BC00392 VJ=100.00  +MOVJ EC00392 VJ=100.00
MOVJ C00393 BC00393 VJ=100.00  +MOVJ EC00393 VJ=100.00
'
END
